// Block: Area02_Messages

DATA_BLOCK Area02_Messages
VERSION : 0.1
   NON_RETAIN
   VAR
      A : Struct
         Msg : Array[1..576] of Bool;
         Hmi : Array[1..36] of Word;
         Ack : Array[1..36] of Word;
      END_STRUCT;
      W : Struct
         Msg : Array[1..384] of Bool;
         Hmi : Array[1..24] of Word;
         Ack : Array[1..24] of Word;
      END_STRUCT;
   END_VAR

BEGIN
   // No initialization required
END_DATA_BLOCK
